FUNCTION_BLOCK CM_DO
VAR_INPUT
	PI_Enable : BOOL;
END_VAR
VAR_OUTPUT
	PO_HighCommand : BOOL;
	PO_LowCommand : BOOL;
END_VAR
VAR_IN_OUT
	Control_data_DO : CM_DO_UDT;
END_VAR

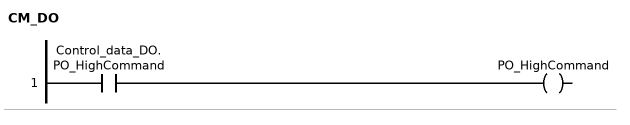
// NETWORK 1
PO_HighCommand := Control_data_DO.PO_HighCommand;

END_FUNCTION_BLOCK

(* stored: Version 1.1.0.1, ProductVersion 3.1.4024.13
   POU CM_DO: Id {b2363562-5ff2-438c-9c32-9788f90e68b9}, SpecialFunc None *)
